% RSLogix 500 project Job 12 Part 2 - Leo Kniffen.RSS, saved by version 10.00.00.00 %
PROJECT "UNTITLED"    % processor: Bul.1763 MicroLogix 1100 Series B %

PROGRAM FILES
  LAD 2   10 rungs

DATA FILES
  O0 OUTPUT  4 elements
  I1 INPUT  6 elements
  S2 STATUS  66 elements
  B3 BINARY  1 elements
  T4 TIMER  1 elements
  C5 COUNTER  1 elements
  R6 CONTROL  1 elements
  N7 INTEGER  1 elements
  F8 FLOAT  1 elements

LADDER 2
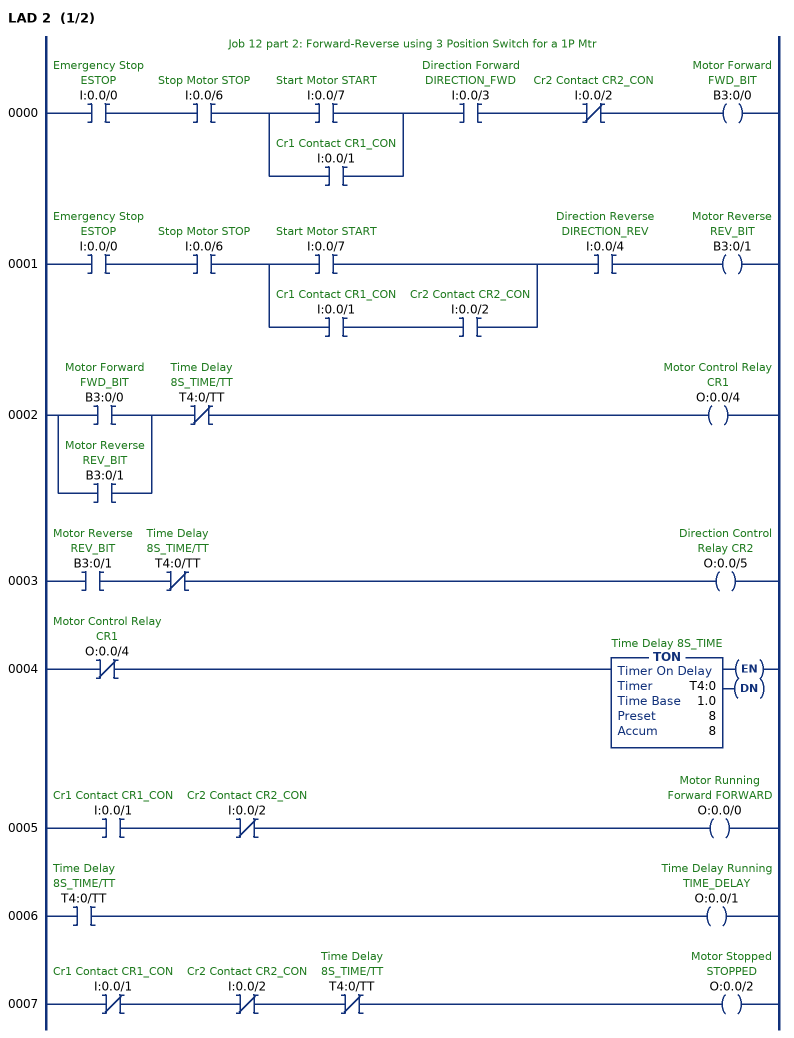
% Rung: 0 %
% Job 12 part 2: Forward-Reverse using 3 Position Switch for a 1P Mtr %
SOR XIC I:0.0/0 XIC I:0.0/6 BST XIC I:0.0/7 NXB XIC I:0.0/1 BND XIC I:0.0/3 XIO I:0.0/2 OTE B3:0/0 EOR
%   I:0.0/0  ESTOP  "Emergency Stop" %
%   I:0.0/6  STOP  "Stop Motor" %
%   I:0.0/7  START  "Start Motor" %
%   I:0.0/1  CR1_CON  "Cr1 Contact" %
%   I:0.0/3  DIRECTION_FWD  "Direction Forward" %
%   I:0.0/2  CR2_CON  "Cr2 Contact" %
%   B3:0/0  FWD_BIT  "Motor Forward" %
% Rung: 1 %
SOR XIC I:0.0/0 XIC I:0.0/6 BST XIC I:0.0/7 NXB XIC I:0.0/1 XIC I:0.0/2 BND XIC I:0.0/4 OTE B3:0/1 EOR
%   I:0.0/0  ESTOP  "Emergency Stop" %
%   I:0.0/6  STOP  "Stop Motor" %
%   I:0.0/7  START  "Start Motor" %
%   I:0.0/1  CR1_CON  "Cr1 Contact" %
%   I:0.0/2  CR2_CON  "Cr2 Contact" %
%   I:0.0/4  DIRECTION_REV  "Direction Reverse" %
%   B3:0/1  REV_BIT  "Motor Reverse" %
% Rung: 2 %
SOR BST XIC B3:0/0 NXB XIC B3:0/1 BND XIO T4:0/TT OTE O:0.0/4 EOR
%   B3:0/0  FWD_BIT  "Motor Forward" %
%   B3:0/1  REV_BIT  "Motor Reverse" %
%   T4:0  8S_TIME  "Time Delay" %
%   O:0.0/4  CR1  "Motor Control Relay" %
% Rung: 3 %
SOR XIC B3:0/1 XIO T4:0/TT OTE O:0.0/5 EOR
%   B3:0/1  REV_BIT  "Motor Reverse" %
%   T4:0  8S_TIME  "Time Delay" %
%   O:0.0/5  CR2  "Direction Control Relay" %
% Rung: 4 %
SOR XIO O:0.0/4 TON T4:0 1.0 8 8 EOR
%   O:0.0/4  CR1  "Motor Control Relay" %
%   T4:0  8S_TIME  "Time Delay" %
% Rung: 5 %
SOR XIC I:0.0/1 XIO I:0.0/2 OTE O:0.0/0 EOR
%   I:0.0/1  CR1_CON  "Cr1 Contact" %
%   I:0.0/2  CR2_CON  "Cr2 Contact" %
%   O:0.0/0  FORWARD  "Motor Running Forward" %
% Rung: 6 %
SOR XIC T4:0/TT OTE O:0.0/1 EOR
%   T4:0  8S_TIME  "Time Delay" %
%   O:0.0/1  TIME_DELAY  "Time Delay Running" %
% Rung: 7 %
SOR XIO I:0.0/1 XIO I:0.0/2 XIO T4:0/TT OTE O:0.0/2 EOR
%   I:0.0/1  CR1_CON  "Cr1 Contact" %
%   I:0.0/2  CR2_CON  "Cr2 Contact" %
%   T4:0  8S_TIME  "Time Delay" %
%   O:0.0/2  STOPPED  "Motor Stopped" %

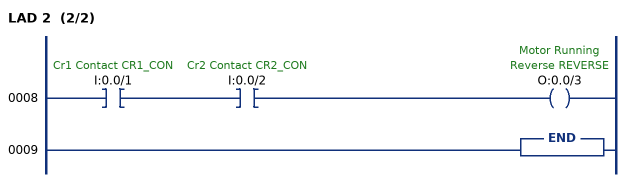
% Rung: 8 %
SOR XIC I:0.0/1 XIC I:0.0/2 OTE O:0.0/3 EOR
%   I:0.0/1  CR1_CON  "Cr1 Contact" %
%   I:0.0/2  CR2_CON  "Cr2 Contact" %
%   O:0.0/3  REVERSE  "Motor Running Reverse" %
% Rung: 9 %
SOR END EOR

DATA TABLE (non-zero values as saved)
DATA T4
% .PRE .ACC %
% T4:0 % 8 8
